// Mitsubishi GX Works2 project: 20150824(from,to消してない)   PLC: Q03UDV

PROGRAM P1
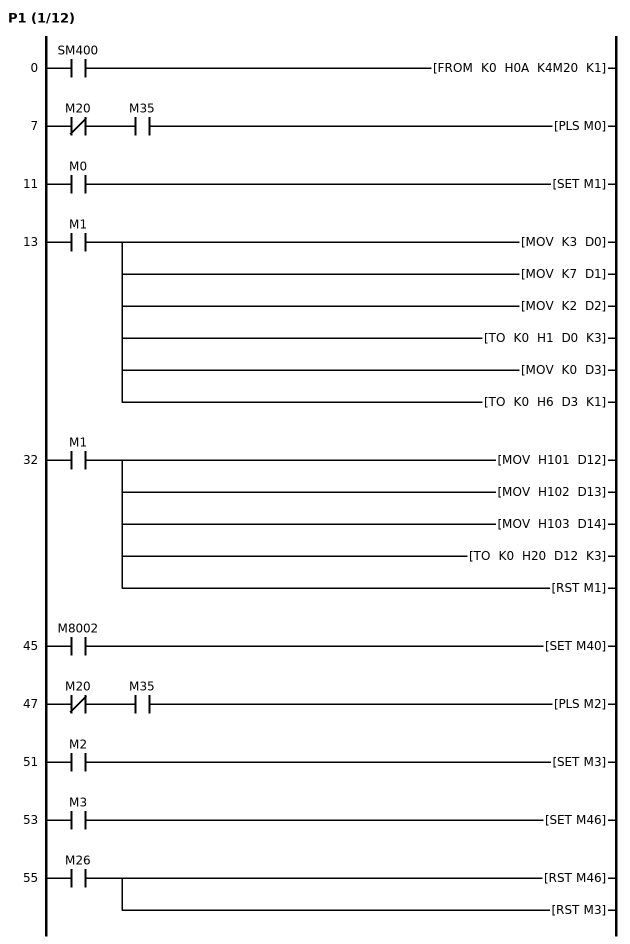
0     LD      SM400
      FROM    K0 H0A K4M20 K1
7     LDI     M20
      AND     M35
      PLS     M0
11    LD      M0
      SET     M1
13    LD      M1
      MOV     K3 D0
      MOV     K7 D1
      MOV     K2 D2
      TO      K0 H1 D0 K3
      MOV     K0 D3
      TO      K0 H6 D3 K1
32    LD      M1
      MOV     H101 D12
      MOV     H102 D13
      MOV     H103 D14
      TO      K0 H20 D12 K3
      RST     M1
45    LD      M8002
      SET     M40
47    LDI     M20
      AND     M35
      PLS     M2
51    LD      M2
      SET     M3
53    LD      M3
      SET     M46
55    LD      M26
      RST     M46
      RST     M3
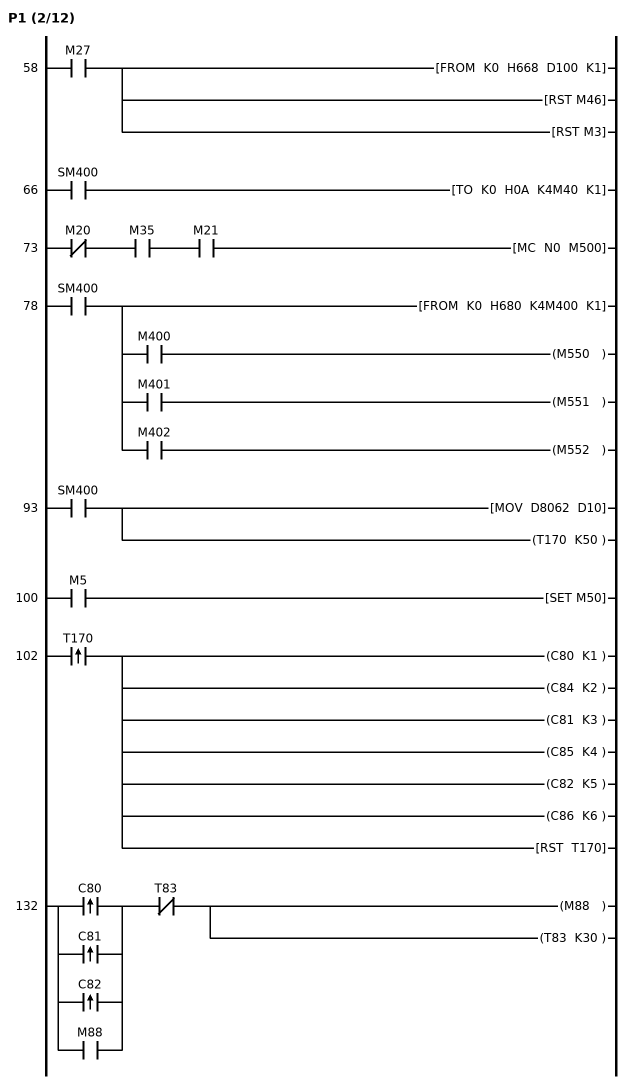
58    LD      M27
      FROM    K0 H668 D100 K1
      RST     M46
      RST     M3
66    LD      SM400
      TO      K0 H0A K4M40 K1
73    LDI     M20
      AND     M35
      AND     M21
      MC      N0 M500
78    LD      SM400
      FROM    K0 H680 K4M400 K1
      MPS
      AND     M400
      OUT     M550
      MRD
      AND     M401
      OUT     M551
      MPP
      AND     M402
      OUT     M552
93    LD      SM400
      MOV     D8062 D10
      OUT     T170 K50
100   LD      M5
      SET     M50
102   LDP     T170
      OUT     C80 K1
      OUT     C84 K2
      OUT     C81 K3
      OUT     C85 K4
      OUT     C82 K5
      OUT     C86 K6
      RST     T170
132   LDP     C80
      ORP     C81
      ORP     C82
      OR      M88
      ANI     T83
      OUT     M88
      OUT     T83 K30
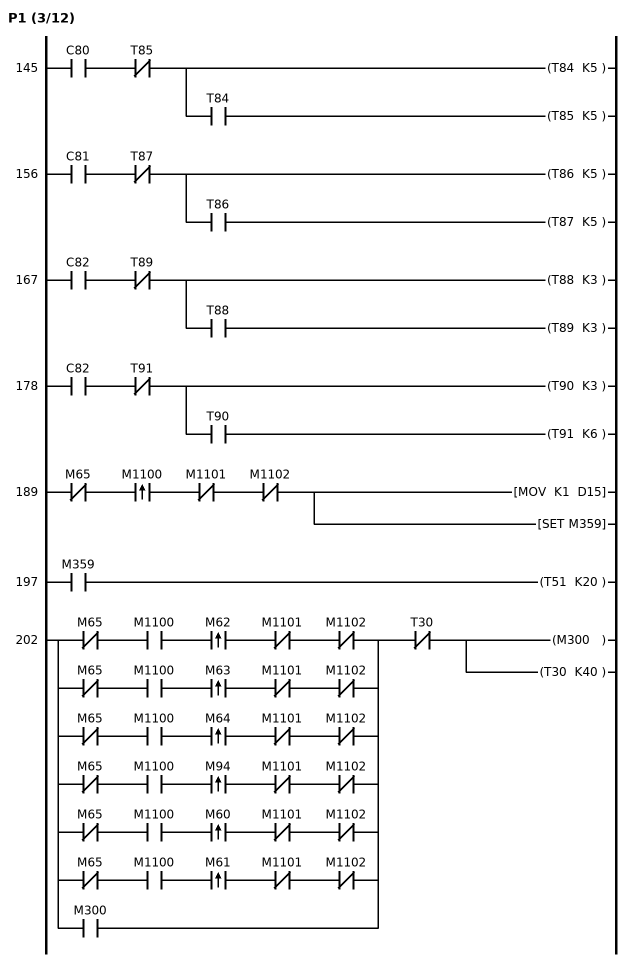
145   LD      C80
      ANI     T85
      OUT     T84 K5
      AND     T84
      OUT     T85 K5
156   LD      C81
      ANI     T87
      OUT     T86 K5
      AND     T86
      OUT     T87 K5
167   LD      C82
      ANI     T89
      OUT     T88 K3
      AND     T88
      OUT     T89 K3
178   LD      C82
      ANI     T91
      OUT     T90 K3
      AND     T90
      OUT     T91 K6
189   LDI     M65
      ANDP    M1100
      ANI     M1101
      ANI     M1102
      MOV     K1 D15
      SET     M359
197   LD      M359
      OUT     T51 K20
202   LDI     M65
      AND     M1100
      ANDP    M62
      ANI     M1101
      ANI     M1102
      LDI     M65
      AND     M1100
      ANDP    M63
      ANI     M1101
      ANI     M1102
      ORB
      LDI     M65
      AND     M1100
      ANDP    M64
      ANI     M1101
      ANI     M1102
      ORB
      LDI     M65
      AND     M1100
      ANDP    M94
      ANI     M1101
      ANI     M1102
      ORB
      LDI     M65
      AND     M1100
      ANDP    M60
      ANI     M1101
      ANI     M1102
      ORB
      LDI     M65
      AND     M1100
      ANDP    M61
      ANI     M1101
      ANI     M1102
      ORB
      OR      M300
      ANI     T30
      OUT     M300
      OUT     T30 K40
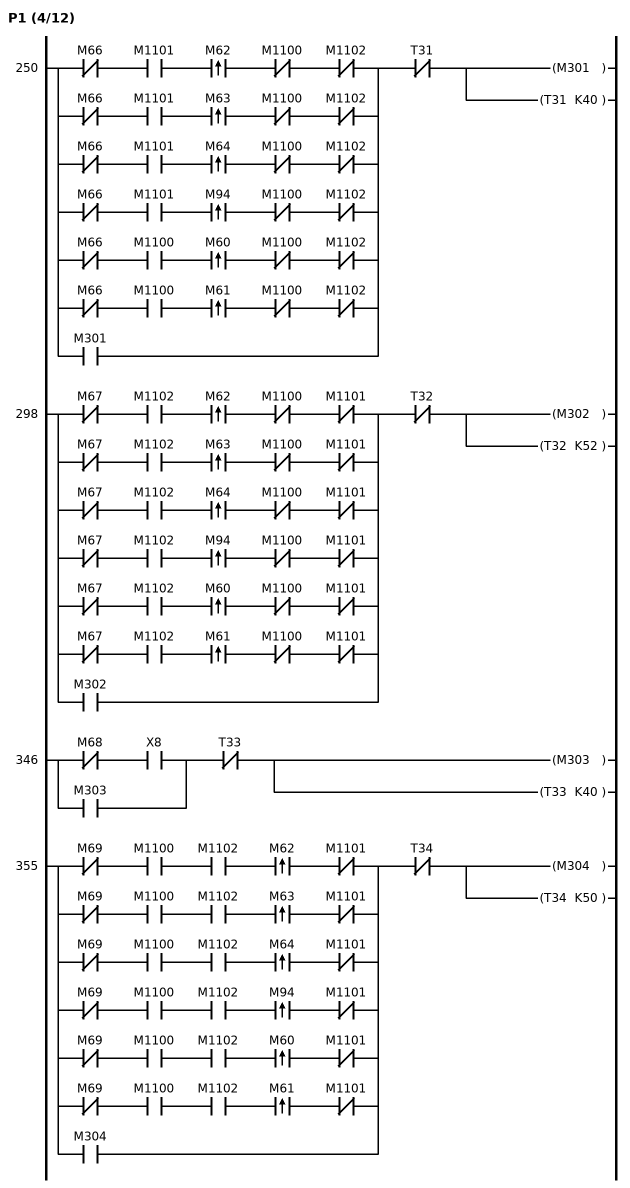
250   LDI     M66
      AND     M1101
      ANDP    M62
      ANI     M1100
      ANI     M1102
      LDI     M66
      AND     M1101
      ANDP    M63
      ANI     M1100
      ANI     M1102
      ORB
      LDI     M66
      AND     M1101
      ANDP    M64
      ANI     M1100
      ANI     M1102
      ORB
      LDI     M66
      AND     M1101
      ANDP    M94
      ANI     M1100
      ANI     M1102
      ORB
      LDI     M66
      AND     M1100
      ANDP    M60
      ANI     M1100
      ANI     M1102
      ORB
      LDI     M66
      AND     M1100
      ANDP    M61
      ANI     M1100
      ANI     M1102
      ORB
      OR      M301
      ANI     T31
      OUT     M301
      OUT     T31 K40
298   LDI     M67
      AND     M1102
      ANDP    M62
      ANI     M1100
      ANI     M1101
      LDI     M67
      AND     M1102
      ANDP    M63
      ANI     M1100
      ANI     M1101
      ORB
      LDI     M67
      AND     M1102
      ANDP    M64
      ANI     M1100
      ANI     M1101
      ORB
      LDI     M67
      AND     M1102
      ANDP    M94
      ANI     M1100
      ANI     M1101
      ORB
      LDI     M67
      AND     M1102
      ANDP    M60
      ANI     M1100
      ANI     M1101
      ORB
      LDI     M67
      AND     M1102
      ANDP    M61
      ANI     M1100
      ANI     M1101
      ORB
      OR      M302
      ANI     T32
      OUT     M302
      OUT     T32 K52
346   LDI     M68
      AND     X8
      OR      M303
      ANI     T33
      OUT     M303
      OUT     T33 K40
355   LDI     M69
      AND     M1100
      AND     M1102
      ANDP    M62
      ANI     M1101
      LDI     M69
      AND     M1100
      AND     M1102
      ANDP    M63
      ANI     M1101
      ORB
      LDI     M69
      AND     M1100
      AND     M1102
      ANDP    M64
      ANI     M1101
      ORB
      LDI     M69
      AND     M1100
      AND     M1102
      ANDP    M94
      ANI     M1101
      ORB
      LDI     M69
      AND     M1100
      AND     M1102
      ANDP    M60
      ANI     M1101
      ORB
      LDI     M69
      AND     M1100
      AND     M1102
      ANDP    M61
      ANI     M1101
      ORB
      OR      M304
      ANI     T34
      OUT     M304
      OUT     T34 K50
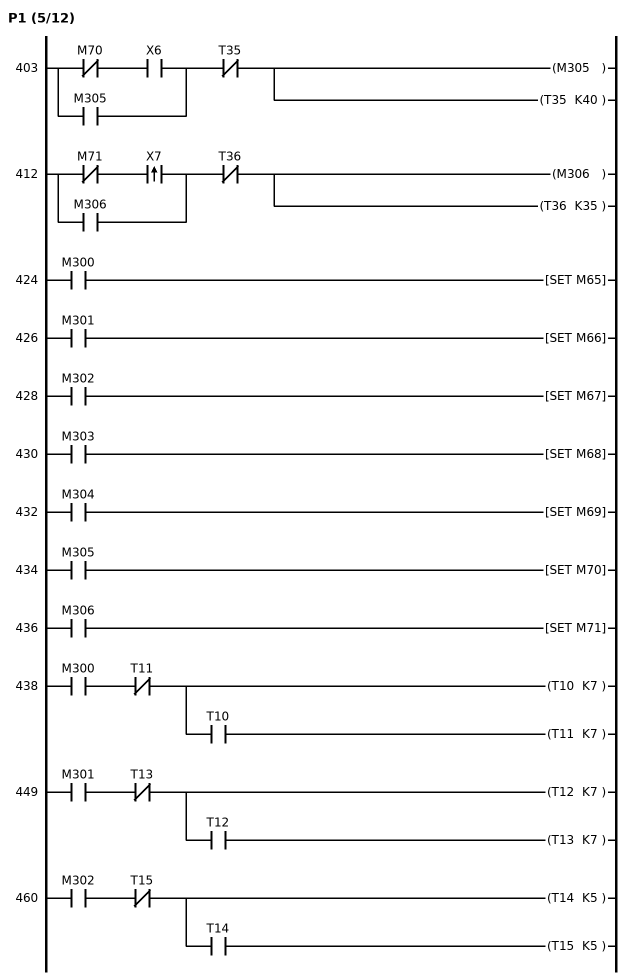
403   LDI     M70
      AND     X6
      OR      M305
      ANI     T35
      OUT     M305
      OUT     T35 K40
412   LDI     M71
      ANDP    X7
      OR      M306
      ANI     T36
      OUT     M306
      OUT     T36 K35
424   LD      M300
      SET     M65
426   LD      M301
      SET     M66
428   LD      M302
      SET     M67
430   LD      M303
      SET     M68
432   LD      M304
      SET     M69
434   LD      M305
      SET     M70
436   LD      M306
      SET     M71
438   LD      M300
      ANI     T11
      OUT     T10 K7
      AND     T10
      OUT     T11 K7
449   LD      M301
      ANI     T13
      OUT     T12 K7
      AND     T12
      OUT     T13 K7
460   LD      M302
      ANI     T15
      OUT     T14 K5
      AND     T14
      OUT     T15 K5
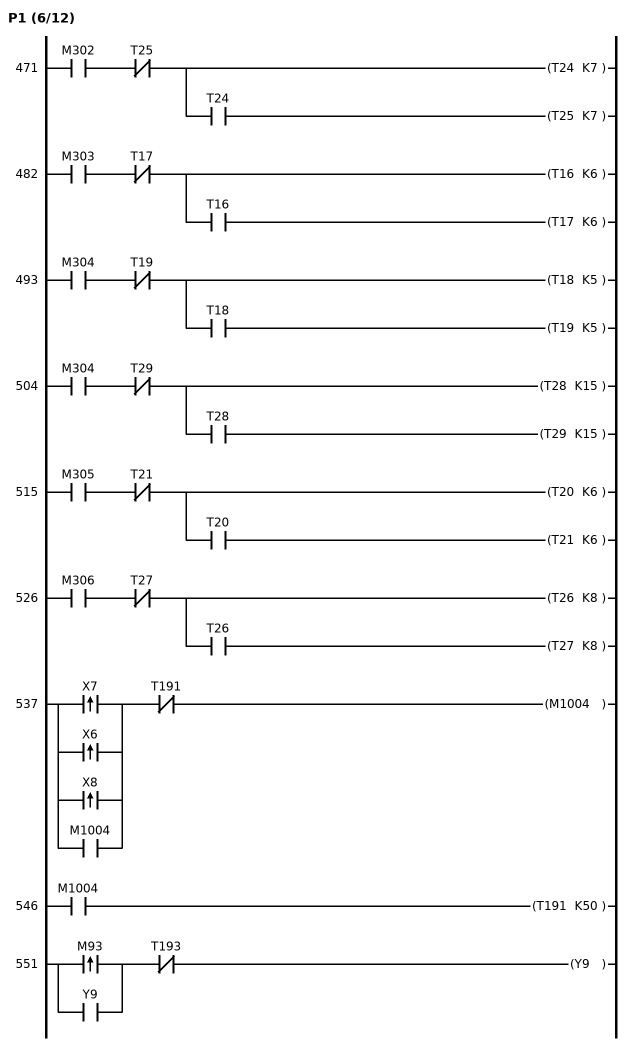
471   LD      M302
      ANI     T25
      OUT     T24 K7
      AND     T24
      OUT     T25 K7
482   LD      M303
      ANI     T17
      OUT     T16 K6
      AND     T16
      OUT     T17 K6
493   LD      M304
      ANI     T19
      OUT     T18 K5
      AND     T18
      OUT     T19 K5
504   LD      M304
      ANI     T29
      OUT     T28 K15
      AND     T28
      OUT     T29 K15
515   LD      M305
      ANI     T21
      OUT     T20 K6
      AND     T20
      OUT     T21 K6
526   LD      M306
      ANI     T27
      OUT     T26 K8
      AND     T26
      OUT     T27 K8
537   LDP     X7
      ORP     X6
      ORP     X8
      OR      M1004
      ANI     T191
      OUT     M1004
546   LD      M1004
      OUT     T191 K50
551   LDP     M93
      OR      Y9
      ANI     T193
      OUT     Y9
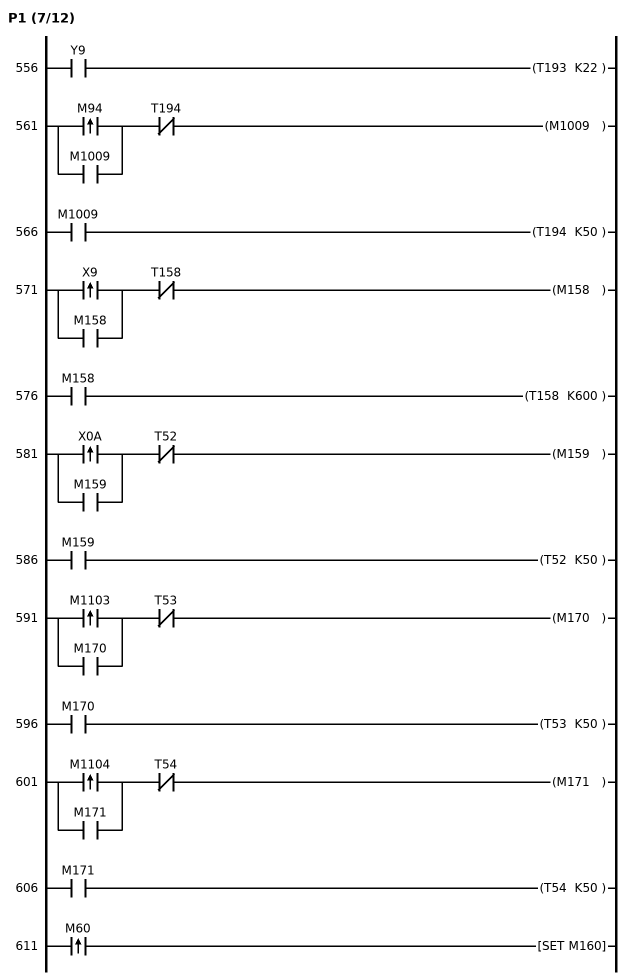
556   LD      Y9
      OUT     T193 K22
561   LDP     M94
      OR      M1009
      ANI     T194
      OUT     M1009
566   LD      M1009
      OUT     T194 K50
571   LDP     X9
      OR      M158
      ANI     T158
      OUT     M158
576   LD      M158
      OUT     T158 K600
581   LDP     X0A
      OR      M159
      ANI     T52
      OUT     M159
586   LD      M159
      OUT     T52 K50
591   LDP     M1103
      OR      M170
      ANI     T53
      OUT     M170
596   LD      M170
      OUT     T53 K50
601   LDP     M1104
      OR      M171
      ANI     T54
      OUT     M171
606   LD      M171
      OUT     T54 K50
611   LDP     M60
      SET     M160
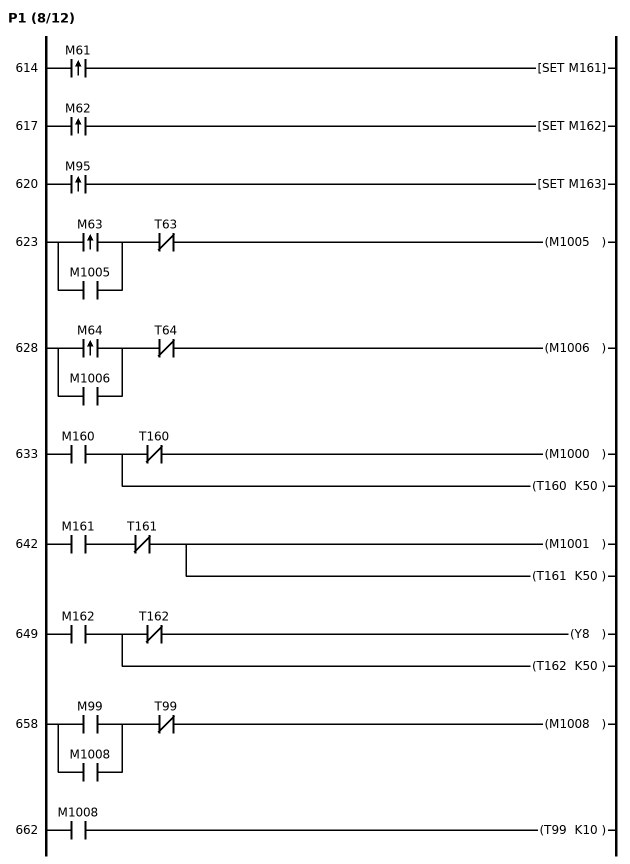
614   LDP     M61
      SET     M161
617   LDP     M62
      SET     M162
620   LDP     M95
      SET     M163
623   LDP     M63
      OR      M1005
      ANI     T63
      OUT     M1005
628   LDP     M64
      OR      M1006
      ANI     T64
      OUT     M1006
633   LD      M160
      MPS
      ANI     T160
      OUT     M1000
      MPP
      OUT     T160 K50
642   LD      M161
      ANI     T161
      OUT     M1001
      OUT     T161 K50
649   LD      M162
      MPS
      ANI     T162
      OUT     Y8
      MPP
      OUT     T162 K50
658   LD      M99
      OR      M1008
      ANI     T99
      OUT     M1008
662   LD      M1008
      OUT     T99 K10
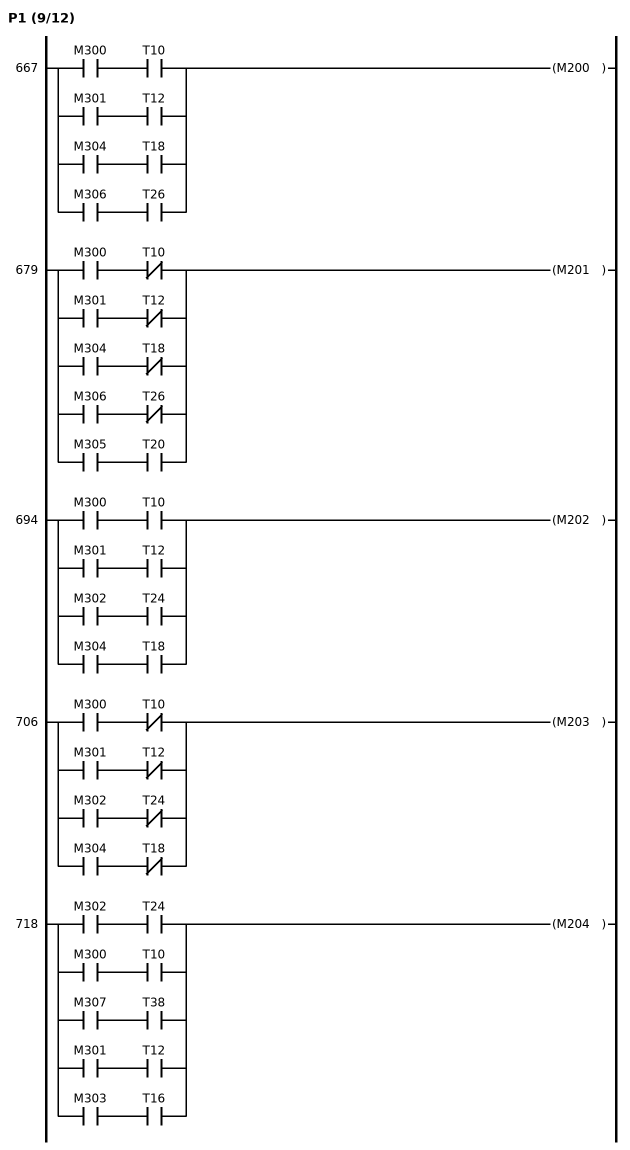
667   LD      M300
      AND     T10
      LD      M301
      AND     T12
      ORB
      LD      M304
      AND     T18
      ORB
      LD      M306
      AND     T26
      ORB
      OUT     M200
679   LD      M300
      ANI     T10
      LD      M301
      ANI     T12
      ORB
      LD      M304
      ANI     T18
      ORB
      LD      M306
      ANI     T26
      ORB
      LD      M305
      AND     T20
      ORB
      OUT     M201
694   LD      M300
      AND     T10
      LD      M301
      AND     T12
      ORB
      LD      M302
      AND     T24
      ORB
      LD      M304
      AND     T18
      ORB
      OUT     M202
706   LD      M300
      ANI     T10
      LD      M301
      ANI     T12
      ORB
      LD      M302
      ANI     T24
      ORB
      LD      M304
      ANI     T18
      ORB
      OUT     M203
718   LD      M302
      AND     T24
      LD      M300
      AND     T10
      ORB
      LD      M307
      AND     T38
      ORB
      LD      M301
      AND     T12
      ORB
      LD      M303
      AND     T16
      ORB
      OUT     M204
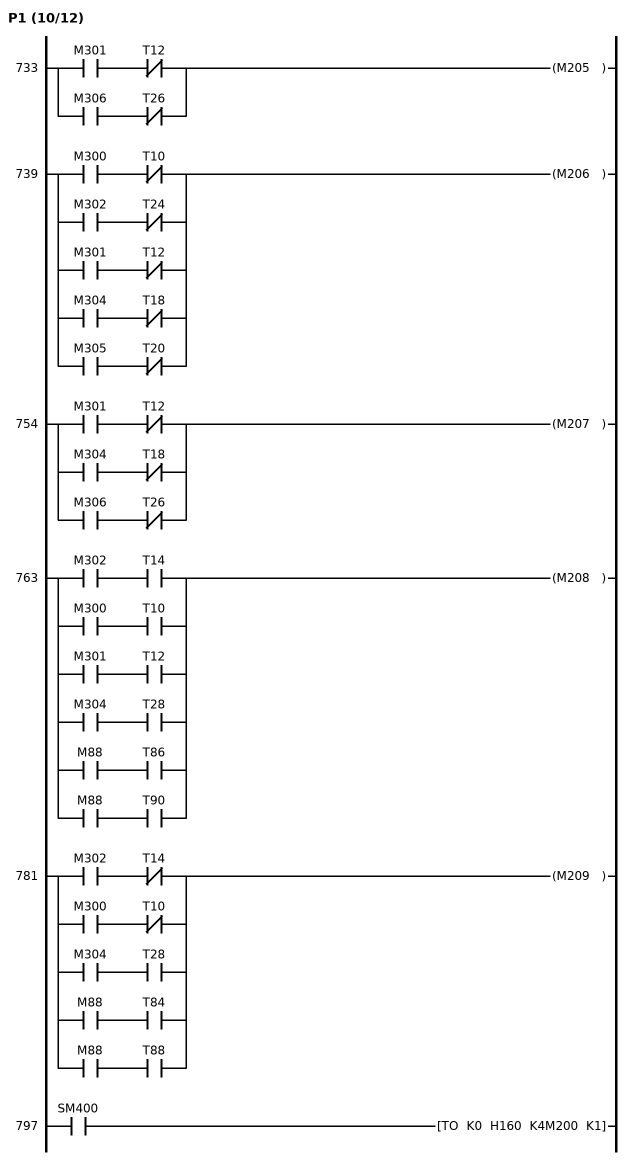
733   LD      M301
      ANI     T12
      LD      M306
      ANI     T26
      ORB
      OUT     M205
739   LD      M300
      ANI     T10
      LD      M302
      ANI     T24
      ORB
      LD      M301
      ANI     T12
      ORB
      LD      M304
      ANI     T18
      ORB
      LD      M305
      ANI     T20
      ORB
      OUT     M206
754   LD      M301
      ANI     T12
      LD      M304
      ANI     T18
      ORB
      LD      M306
      ANI     T26
      ORB
      OUT     M207
763   LD      M302
      AND     T14
      LD      M300
      AND     T10
      ORB
      LD      M301
      AND     T12
      ORB
      LD      M304
      AND     T28
      ORB
      LD      M88
      AND     T86
      ORB
      LD      M88
      AND     T90
      ORB
      OUT     M208
781   LD      M302
      ANI     T14
      LD      M300
      ANI     T10
      ORB
      LD      M304
      AND     T28
      ORB
      LD      M88
      AND     T84
      ORB
      LD      M88
      AND     T88
      ORB
      OUT     M209
797   LD      SM400
      TO      K0 H160 K4M200 K1
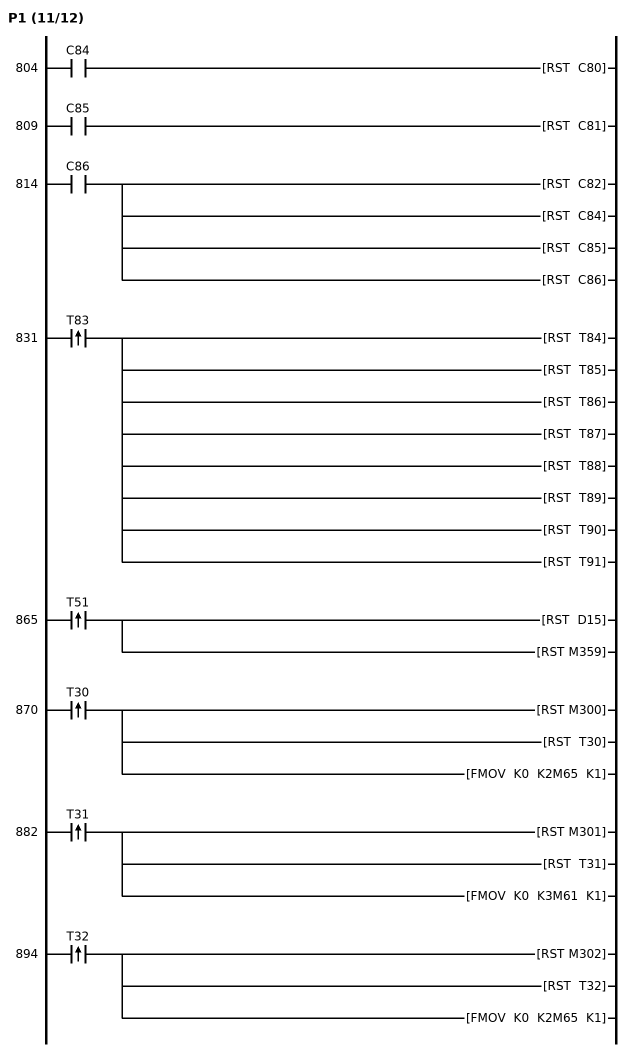
804   LD      C84
      RST     C80
809   LD      C85
      RST     C81
814   LD      C86
      RST     C82
      RST     C84
      RST     C85
      RST     C86
831   LDP     T83
      RST     T84
      RST     T85
      RST     T86
      RST     T87
      RST     T88
      RST     T89
      RST     T90
      RST     T91
865   LDP     T51
      RST     D15
      RST     M359
870   LDP     T30
      RST     M300
      RST     T30
      FMOV    K0 K2M65 K1
882   LDP     T31
      RST     M301
      RST     T31
      FMOV    K0 K3M61 K1
894   LDP     T32
      RST     M302
      RST     T32
      FMOV    K0 K2M65 K1
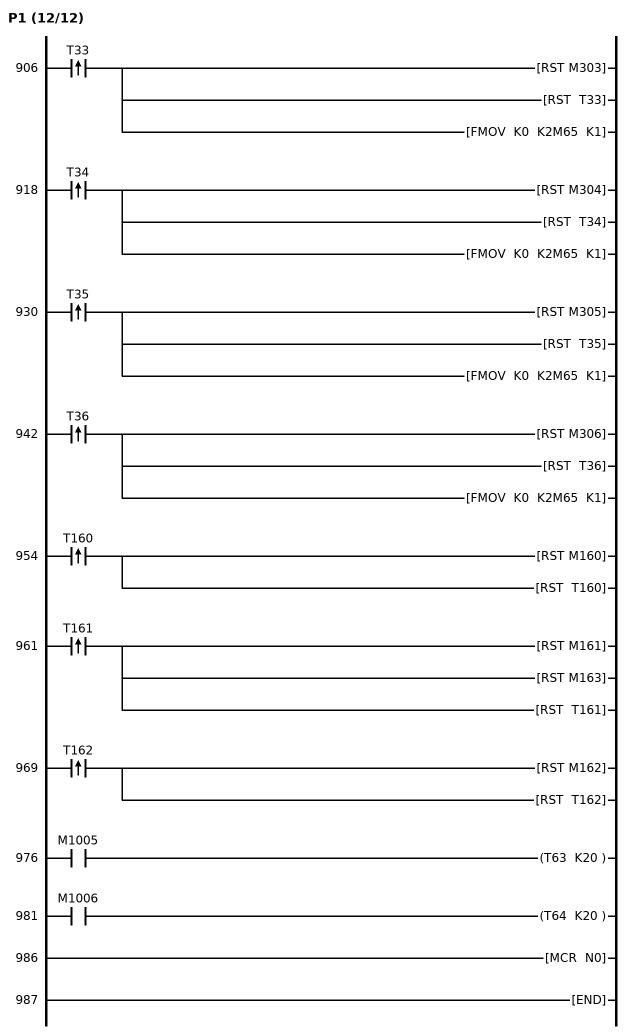
906   LDP     T33
      RST     M303
      RST     T33
      FMOV    K0 K2M65 K1
918   LDP     T34
      RST     M304
      RST     T34
      FMOV    K0 K2M65 K1
930   LDP     T35
      RST     M305
      RST     T35
      FMOV    K0 K2M65 K1
942   LDP     T36
      RST     M306
      RST     T36
      FMOV    K0 K2M65 K1
954   LDP     T160
      RST     M160
      RST     T160
961   LDP     T161
      RST     M161
      RST     M163
      RST     T161
969   LDP     T162
      RST     M162
      RST     T162
976   LD      M1005
      OUT     T63 K20
981   LD      M1006
      OUT     T64 K20
986   MCR     N0
987   END
END_PROGRAM

PROGRAM P2
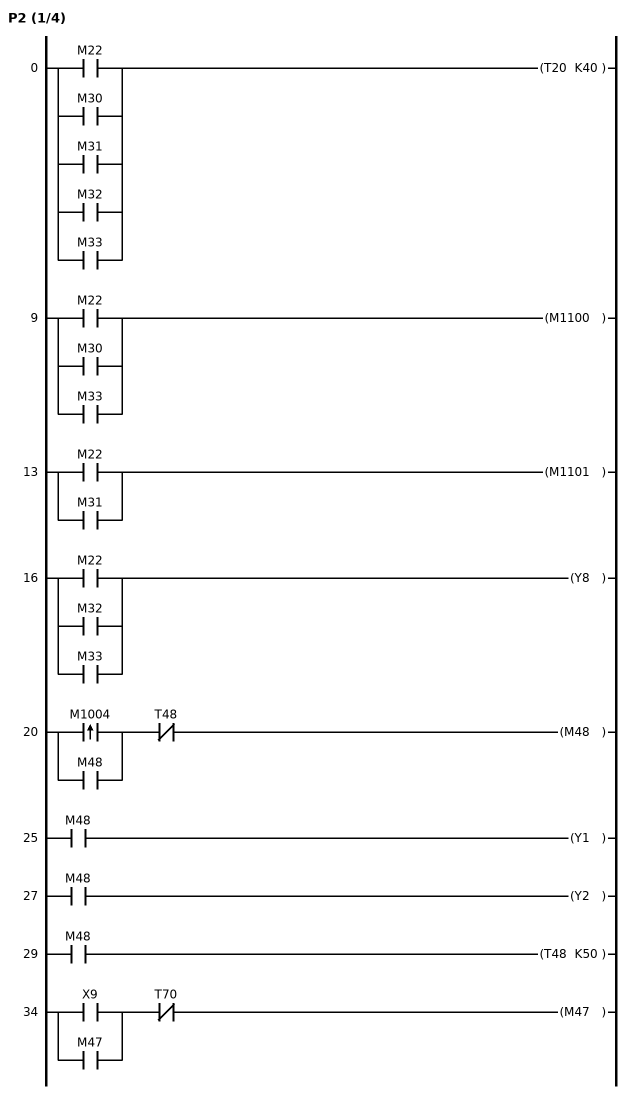
0     LD      M22
      OR      M30
      OR      M31
      OR      M32
      OR      M33
      OUT     T20 K40
9     LD      M22
      OR      M30
      OR      M33
      OUT     M1100
13    LD      M22
      OR      M31
      OUT     M1101
16    LD      M22
      OR      M32
      OR      M33
      OUT     Y8
20    LDP     M1004
      OR      M48
      ANI     T48
      OUT     M48
25    LD      M48
      OUT     Y1
27    LD      M48
      OUT     Y2
29    LD      M48
      OUT     T48 K50
34    LD      X9
      OR      M47
      ANI     T70
      OUT     M47
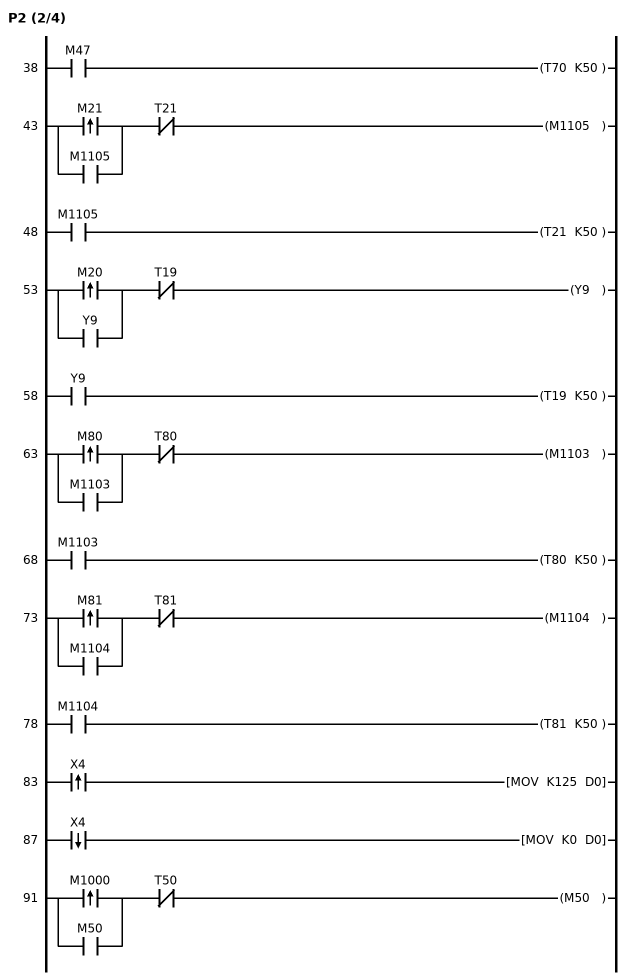
38    LD      M47
      OUT     T70 K50
43    LDP     M21
      OR      M1105
      ANI     T21
      OUT     M1105
48    LD      M1105
      OUT     T21 K50
53    LDP     M20
      OR      Y9
      ANI     T19
      OUT     Y9
58    LD      Y9
      OUT     T19 K50
63    LDP     M80
      OR      M1103
      ANI     T80
      OUT     M1103
68    LD      M1103
      OUT     T80 K50
73    LDP     M81
      OR      M1104
      ANI     T81
      OUT     M1104
78    LD      M1104
      OUT     T81 K50
83    LDP     X4
      MOV     K125 D0
87    LDF     X4
      MOV     K0 D0
91    LDP     M1000
      OR      M50
      ANI     T50
      OUT     M50
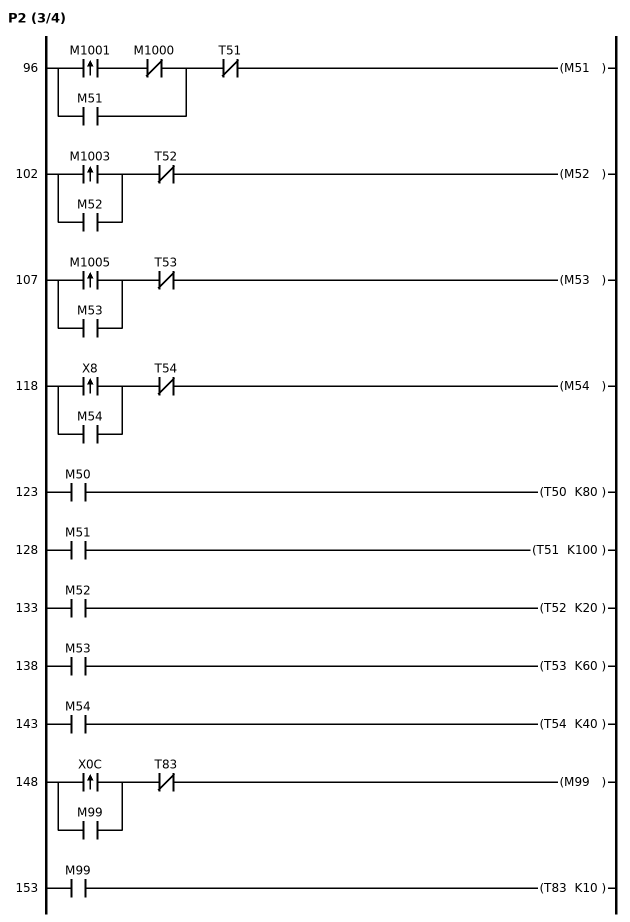
96    LDP     M1001
      ANI     M1000
      OR      M51
      ANI     T51
      OUT     M51
102   LDP     M1003
      OR      M52
      ANI     T52
      OUT     M52
107   LDP     M1005
      OR      M53
      ANI     T53
      OUT     M53
118   LDP     X8
      OR      M54
      ANI     T54
      OUT     M54
123   LD      M50
      OUT     T50 K80
128   LD      M51
      OUT     T51 K100
133   LD      M52
      OUT     T52 K20
138   LD      M53
      OUT     T53 K60
143   LD      M54
      OUT     T54 K40
148   LDP     X0C
      OR      M99
      ANI     T83
      OUT     M99
153   LD      M99
      OUT     T83 K10
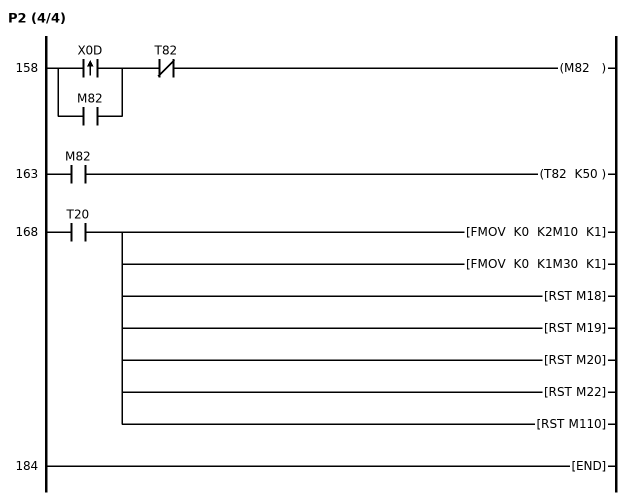
158   LDP     X0D
      OR      M82
      ANI     T82
      OUT     M82
163   LD      M82
      OUT     T82 K50
168   LD      T20
      FMOV    K0 K2M10 K1
      FMOV    K0 K1M30 K1
      RST     M18
      RST     M19
      RST     M20
      RST     M22
      RST     M110
184   END
END_PROGRAM
